{attribute addProperty BoxType "KL1904"}
{attribute addProperty Id "Safety_InAT %I*ARRAY[0..5] OF BYTE000Safety_OutAT %Q*ARRAY[0..5] OF BYTE000"}
{attribute addProperty CRC "3630243302"}
{attribute addProperty SizeInBites "0"}
{attribute addProperty SizeInBytes "0"}
TYPE Channel_D8611DE6 :
STRUCT
	{attribute addProperty Name "Safety_In"}
	Safety_In AT %I* : ARRAY[0..5] OF BYTE;
	{attribute addProperty Name "Safety_Out"}
	Safety_Out AT %Q* : ARRAY[0..5] OF BYTE;
END_STRUCT
END_TYPE

(* stored: Version 1.2.0.0, ProductVersion 3.1.4024.9
   DUT Channel_D8611DE6: Id {dac06f40-0cc0-42b9-a63c-ef9de8f8665e} *)
